									stSlideNest.State				:= E_SlideNest_State.READY;									
									bNestLeft						:= FALSE;
																	
								END_IF
	
	
	E_SlideNest_State.READY:
	
								IF stSlideNest.CMD.bExecute AND 	stSlideNest.CMD.SlideCylinderCMD.MoveRight	THEN

									stSlideNest.State				:= E_SlideNest_State.MOVE_RIGHT;
									
								ELSIF stSlideNest.CMD.bExecute AND 	stSlideNest.CMD.SlideCylinderCMD.MoveLeft	THEN
									
									stSlideNest.State				:= E_SlideNest_State.MOVE_LEFT;									
																		
								END_IF
	

	E_SlideNest_State.MOVE_RIGHT:
	
								bNestRight							:= TRUE;
								
								IF bNestInRightPos	THEN
									
									stSlideNest.State				:= E_SlideNest_State.DONE;
								
								END_IF
								
	E_SlideNest_State.MOVE_LEFT:
	
								bNestLeft							:= TRUE;
								
								IF bNestInLeftPos THEN
									
									stSlideNest.State				:= E_SlideNest_State.DONE;
								
								END_IF
								
	E_SlideNest_State.DONE:
	
	
								IF stSlideNest.CMD.bAcknowledge THEN
									
									stSlideNest.CMD.bAcknowledge	:= FALSE;
									stSlideNest.State				:= E_SlideNest_State.RESET;
								
								END_IF
	
	
	E_SlideNest_State.RESET:	
	
								bNestRight							:= FALSE;
								bNestLeft							:= FALSE;
								
								IF NOT stSlideNest.CMD.bAbort AND NOT stSlideNest.CMD.bEndCycle THEN
									
									stSlideNest.State				:= E_SlideNest_State.READY;
									
								ELSE stSlideNest.State			:= E_SlideNest_State.ABORTED;
								END_IF
									

ELSE stSlideNest.State		:= E_SlideNest_State.ABORTED;
	
END_CASE
/////////////////////////////////////////////////////////////////////////////////////STATUS/////////////////////////////////////////////////////////////////////////////////////

stSlideNest.Status.bBusy			:= 	stSlideNest.State	= E_SlideNest_State.MOVE_RIGHT OR
										stSlideNest.State	= E_SlideNest_State.MOVE_LEFT OR 
										stSlideNest.State	= E_SlideNest_State.STOPPING;
								
stSlideNest.Status.bDone			:=	stSlideNest.State	= E_SlideNest_State.DONE;

stSlideNest.Status.bReady			:= 	stSlideNest.State	= E_SlideNest_State.READY;

stSlideNest.Status.bStopped		:= 	NOT stSlideNest.Status.bBusy;
END_ACTION

ACTION b_ACT_IO_B:

bNestInLeftPos									:= dw_T08_EL1809.iSlideNestRetracted;
bNestInRightPos									:= dw_T08_EL1809.iSlideNestExtended; 

dw_T09_EL2809.qExtendSlideNest					:= bNestRight OR bSlideNestRight;	
dw_T09_EL2809.qRetractSlideNest					:= bNestLeft OR bSlideNestLeft;

bProcessCylinderUp								:= stTwinSAFE.qProcessCylinderRetracted;
END_ACTION

ACTION d_ACT_Set_Events_Station_4B:
//IMMEDIATE FAULTS

stStationEvents[4].aEvents[0].bEventTimer( IN :=  (bNestRight OR bSlideNestLeft) AND NOT bNestInLeftPos, PT := T#5S);
stStationEvents[4].aEvents[0].bFault						:= TRUE;
stStationEvents[4].aEvents[0].bEventFlag					:= stStationEvents[4].aEvents[0].bEventTimer.Q;
stStationEvents[4].aEvents[0].bEventText					:= 'Process Door extend timeout';
stStationEvents[4].aEvents[0].sSolution						:= 'Check cylinder, neumatic connections and sensors';

stStationEvents[4].aEvents[1].bEventTimer( IN :=  (bNestLeft OR bSlideNestRight) AND NOT bNestInRightPos, PT := T#5S);
stStationEvents[4].aEvents[1].bFault						:= TRUE;
stStationEvents[4].aEvents[1].bEventFlag					:= stStationEvents[4].aEvents[1].bEventTimer.Q;
stStationEvents[4].aEvents[1].bEventText					:= 'Process Door Retract timeout';
stStationEvents[4].aEvents[1].sSolution						:= 'Check cylinder, neumatic connections and sensors';
END_ACTION

END_PROGRAM

// ---- POUs/A_MASTER/A_2_PRG_MachineCtrl.TcPOU
PROGRAM A_2_PRG_MachineCtrl
VAR
/////////////////////////////////////////////////////////////////////////////////////TIMERS & TRIGGERS/////////////////////////////////////////////////////////////////////////////////////

	tonSys_Init					: Tc2_Standard.TON:=(PT:=T#1S);
	tonSys_InitTimeout			: Tc2_Standard.TON:=(PT:=T#15S);					
	tonFirstAutoCycle			: Tc2_Standard.TON:=(PT:=T#500MS);
	tonStopped					: TON := (PT := T#500MS);
	
/////////////////////////////////////////////////////////////////////////////////////PROCESS CYCLE/////////////////////////////////////////////////////////////////////////////////////	
	
	eCycleState					: E_General_ProcessCycle;
	tonCMD_Done					: TON;
	tonResetAllCMD				: TON;
	tonExecute					: TON;
	tonSave_Data				: TON;
	tonWriteToCsv				: TON;
	rFirstAutoCycle				: R_TRIG;
	
	bStartProcessCondition		: BOOL;
	bLeakTestDoneFlag			: BOOL;
	bHeightTestDoneFlag			: BOOL;
	i							: INT;

	tonGettingResults			: TON;
	ctuRejectPart				: CTU;
	
	tonProcessCylinderDelay		: TON;
	tonSealing					: TON;
	
	tonCylinderDwell			: TON; //Renan added - Buglist n13 - 08Jul26
	
	

/////////////////////////////////////////////////////////////////////////////////////I/O/////////////////////////////////////////////////////////////////////////////////////	

	bSlideNestNotHomed			: BOOL;
	bPartPresentNest1			: BOOL;
	bPartPresentNest2			: BOOL;
	rRejectSensor				: R_TRIG;
	bTwoHandsSignal				: BOOL;
	tonTwoHandsSignal			: TON;
	
	bProcessedPart				: ARRAY[0..1] OF BOOL;
	fProcessedPart				: ARRAY[0..1] OF F_TRIG;
	
		(* Renan Added - Buglist n6 - 08Jul26 *)
	bNest1StartOK				: BOOL;
	bNest2StartOK				: BOOL;
	bCycleHasFailure 			: BOOL;
	bCycleAllProcessedPass		: BOOL;
	(*\Renan Added - Buglist n6 - 08Jul26 *)
	
	bPuckLockerReadyToStart		: BOOL; (* Renan Added - Puck Locker Bug - 08Jul26 *)
	nPucksToRelease 			: USINT;(* Renan Added - Puck Locker Bug - 08Jul26 *)
	bPuckLockerEnable       	: BOOL; (* Renan added - Puck Locker Bug - 10Jul26*)
	bTest						: BOOL;
	
	bBottomSealer				: BOOL;
	bTopSealer					: BOOL;
	
	
END_VAR

/////////////////////////////////////////////////////////////////////////////////////GENERAL/////////////////////////////////////////////////////////////////////////////////////
a_ACT_MachineStatus();
b_ACT_ProcessCycle();
d_ACT_IO();

ACTION a_ACT_MachineStatus:
/////////////////////////////////////////////////////////////////////////////////////Utilities/////////////////////////////////////////////////////////////////////////////////////
tonSys_Init(IN:=stMachineStatus.bInitialising);
tonSys_InitTimeout(IN:=stMachineStatus.bInitialising);
tonSafety( IN := stMachineStatus.eMachineState = E_MachineState.SAFETY, PT := T#10S);
tonStopped(IN := stMachineStatus.eMachineState = E_MachineState.STOPPED);
	
	IF stMachineStatus.eMachineState <> E_MachineState.SYSTEM_AUTO_CYCLE AND 
		stMachineStatus.eMachineState <> E_MachineState.SYSTEM_INITIALISING THEN
		
		sMachineMessage									:= '';			
		
	END_IF
	
	IF (stMachineStatus.eMachineState = E_MachineState.STOPPED)  OR 
		(stMachineStatus.eMachineState = E_MachineState.STOPPING) THEN
		
		stTwinSAFE.iMachineStopped						:= TRUE;
		stTwinSAFE.iRunSafety							:= FALSE;
	
	ELSIF (stMachineStatus.eMachineState = E_MachineState.SAFETY) OR (stMachineStatus.eMachineState = E_MachineState.SYSTEM_INITIALISING) OR 
		(stMachineStatus.eMachineState = E_MachineState.SYSTEM_READY_TO_START) OR (stMachineStatus.eMachineState = E_MachineState.SYSTEM_AUTO_CYCLE) 
		OR (stMachineStatus.eMachineState = E_MachineState.MANUAL_MODE)THEN

		stTwinSAFE.iRunSafety							:= TRUE;
		stTwinSAFE.iMachineStopped						:= FALSE;
	
	ELSE stTwinSAFE.iMachineStopped						:= FALSE;
		stTwinSAFE.iRunSafety							:= FALSE;
		
	END_IF
	
	IF stMachineStatus.eMachineState = E_MachineState.SAFETY THEN
		
		stTwinSAFE.iInitSafety							:= TRUE;
		
	ELSE stTwinSAFE.iInitSafety							:= FALSE;
		
	END_IF

/////////////////////////////////////////////////////////////////////////////////////CONDITIONS/////////////////////////////////////////////////////////////////////////////////////
				IF NOT stMasterCtrl.bNoFault THEN
					stMachineStatus.eMachineState 		:= E_MachineState.FAULT;
				END_IF
				
				IF stMachineStatus.eMachineState		= E_MachineState.STOPPING OR
				stMachineStatus.eMachineState			= E_MachineState.FAULT THEN
					
					stSlideNest.CMD.bAbort				:= TRUE;	
					stLeakTesters.CMD.bAbort			:= TRUE;	
					stHeightTests.CMD.bAbort			:= TRUE;
					stProcessCylinder.CMD.bAbort		:= TRUE;
					stProcessDoor.CMD.bAbort			:= TRUE;
				
					stSlideNest.CMD.bEnable				:= FALSE;	
					stLeakTesters.CMD.bEnable			:= FALSE;	
					stHeightTests.CMD.bEnable			:= FALSE;
					stProcessCylinder.CMD.bEnable		:= FALSE;
					stProcessDoor.CMD.bEnable			:= FALSE;
					
				END_IF
				
				IF 	stButtonsLamps.bResetButtonFallingEdge THEN
					stSlideNest.CMD.bReset				:= TRUE;	
					stLeakTesters.CMD.bReset			:= TRUE;	
					stHeightTests.CMD.bReset			:= TRUE;
					stProcessCylinder.CMD.bReset		:= TRUE;
					stProcessDoor.CMD.bReset			:= TRUE;
				ELSE 
					stSlideNest.CMD.bReset				:= FALSE;	
					stLeakTesters.CMD.bReset			:= FALSE;	
					stHeightTests.CMD.bReset			:= FALSE;
					stProcessCylinder.CMD.bReset		:= FALSE;
					stProcessDoor.CMD.bReset			:= FALSE;
				END_IF	

				IF 	NOT (stMachineStatus.eMachineState = E_MachineState.MANUAL_MODE) THEN
					
					stSlideNest.CMD.bManualMode				:=FALSE;
					stLeakTesters.CMD.bManualMode			:=FALSE;
					stHeightTests.CMD.bManualMode			:=FALSE;
					stProcessCylinder.CMD.bManualMode		:=FALSE;
					stProcessDoor.CMD.bManualMode			:=FALSE;
					
				END_IF
				
				IF stMachineStatus.eMachineState = E_MachineState.SYSTEM_POWER_UP THEN
					
					bReadAMSNetID							:= TRUE;
				
				ELSE 
					
					bReadAMSNetID							:= FALSE;
					
				END_IF
				
				IF stMachineStatus.eMachineState		= E_MachineState.FAULT THEN
					
					bOpenDoorCycleFault						:= TRUE;
					
				ELSE bOpenDoorCycleFault					:= FALSE;
					
				END_IF
				
/////////////////////////////////////////////////////////////////////////////////////MACHINE CONTROL/////////////////////////////////////////////////////////////////////////////////////

CASE stMachineStatus.eMachineState OF

E_MachineState.SYSTEM_POWER_UP: 		

				fbGetLocalAMSNetID.bExecute				:= TRUE;
				bLightsOnOff							:= TRUE;
				IF tonSystemPowerUP.Q THEN
						stMachineStatus.eMachineState 	:= E_MachineState.STOPPED;//
				END_IF
	
E_MachineState.STOPPED:		

				stTwinSAFE.iRunSafety					:= FALSE;				

				IF stMasterCtrl.bNoFault   AND NOT stMasterCtrl.bCycleStopRequest AND ftrigButton[3].Q AND tonStopped.Q THEN
						stMachineStatus.eMachineState 	:= E_MachineState.SAFETY;//
				ELSIF NOT stMasterCtrl.bNoFault    THEN	
					stMachineStatus.eMachineState 		:= E_MachineState.FAULT;		
				END_IF	

E_MachineState.SAFETY:

				GVL_IO.dw_T09_EL2809.qOpenProcessDoor   := TRUE; // Thays added - Buglist n1 - 08Jul26
				stTwinSAFE.iRunSafety					:= TRUE;
				
				IF stTwinSAFE.qSafetyOk THEN
					
					stMachineStatus.eMachineState		:= E_MachineState.SYSTEM_INITIALISING;
					
				ELSIF stButtonsLamps.bStopButtonFallingEdge OR  
				stMasterCtrl.bCycleStopRequest OR tonSys_InitTimeout.Q  THEN
				
					stMachineStatus.eMachineState 		:= E_MachineState.STOPPING;	
					
				ELSIF NOT stMasterCtrl.bNoFault THEN		
					
					stMachineStatus.eMachineState 		:= E_MachineState.FAULT;
	
				END_IF
								

E_MachineState.SYSTEM_INITIALISING:		
					
					
				stSlideNest.CMD.bAbort					:= FALSE;	
				stLeakTesters.CMD.bAbort				:= FALSE;	
				stHeightTests.CMD.bAbort				:= FALSE;
				stProcessCylinder.CMD.bAbort			:= FALSE;
				stProcessDoor.CMD.bAbort				:= FALSE;	

				IF ( NOT stTwinSAFE.qProcessCylinderRetracted OR bSlideNestNotHomed) AND NOT bProcessDoorClosed THEN
						
						sMachineMessage					:= 'trigger both safety buttons to reset machine';
						
						IF bTwoHandsSignal  THEN
							
							tonSys_InitTimeout.IN		:= TRUE;	
							stLeakTesters.CMD.bEnable	:= TRUE;	
							stHeightTests.CMD.bEnable	:= TRUE;
							stProcessCylinder.CMD.bEnable:= TRUE;
							stProcessDoor.CMD.bEnable	:= TRUE;
							stSlideNest.CMD.bEnable		:= TRUE;
							sMachineMessage				:= '';
							
						END_IF
				ELSIF stTwinSAFE.qProcessCylinderRetracted AND dw_T08_EL1809.iSlideNestRetracted THEN
					
					stSlideNest.CMD.bEnable				:= TRUE;	
					stLeakTesters.CMD.bEnable			:= TRUE;	
					stHeightTests.CMD.bEnable			:= TRUE;
					stProcessCylinder.CMD.bEnable		:= TRUE;
					stProcessDoor.CMD.bEnable			:= TRUE;				
				
				END_IF
				
				IF stMasterCtrl.bAllStationsReady  THEN 
					stMachineStatus.eMachineState		:= E_MachineState.SYSTEM_READY_TO_START;
				ELSIF stButtonsLamps.bStopButtonFallingEdge OR  
				stMasterCtrl.bCycleStopRequest OR tonSys_InitTimeout.Q  THEN
					stMachineStatus.eMachineState 		:= E_MachineState.STOPPING;	
				ELSIF NOT stMasterCtrl.bNoFault THEN		
					stMachineStatus.eMachineState 		:= E_MachineState.FAULT;
				END_IF
			
					
E_MachineState.SYSTEM_READY_TO_START:	

				IF 	 stButtonsLamps.bStartButtonFallingEdge AND stMasterCtrl.bAllStationsReady  THEN
					stMachineStatus.eMachineState 		:= E_MachineState.SYSTEM_AUTO_CYCLE;
				ELSIF NOT stMasterCtrl.bAllStationsReady OR stMasterCtrl.bCycleStopRequest THEN
					stMachineStatus.eMachineState 		:= E_MachineState.STOPPING;		
				ELSIF NOT stMasterCtrl.bNoFault THEN	
					stMachineStatus.eMachineState 		:= E_MachineState.FAULT;
				ELSIF GVL_Master.stMasterCTRL.bManualModeRequest AND stMasterCtrl.bNoFault THEN
					stMachineStatus.eMachineState 		:= E_MachineState.MANUAL_MODE;
				END_IF

				

E_MachineState.SYSTEM_AUTO_CYCLE:		

				
				IF  stMasterCtrl.bCycleStopRequest AND (eCycleState = E_General_ProcessCycle.IDLE) THEN
	
					stMachineStatus.eMachineState 		:= E_MachineState.STOPPING;
				
				ELSIF stMasterCtrl.bCycleStopRequest AND NOT (eCycleState = E_General_ProcessCycle.IDLE) THEN					
				
					sMachineMessage						:= 'Ending  Cycle';
				
				ELSIF NOT stMasterCtrl.bNoFault THEN	
					stMachineStatus.eMachineState 		:= E_MachineState.FAULT;
				END_IF
				

E_MachineState.STOPPING:	

				
				IF stMasterCtrl.bAllStationsStopped THEN
					stMachineStatus.eMachineState 		:= E_MachineState.STOPPED;
				ELSIF NOT stMasterCtrl.bNoFault THEN	
					stMachineStatus.eMachineState 		:= E_MachineState.FAULT;					
				END_IF
				
				stTwinSAFE.iRunSafety					:= FALSE;	

E_MachineState.FAULT:	
				
				GVL_IO.dw_T09_EL2809.qOpenProcessDoor   :=TRUE; // Thays added - Buglist n1 - 08Jul26

				IF stMasterCtrl.bNoFault	THEN
					stMachineStatus.eMachineState		:= E_MachineState.STOPPED;		
				END_IF
				
				stTwinSAFE.iRunSafety					:= FALSE;	

E_MachineState.MANUAL_MODE:

				IF stButtonsLamps.bStopButtonFallingEdge OR NOT GVL_Master.stMasterCTRL.bManualModeRequest THEN
					stMachineStatus.eMachineState 		:= E_MachineState.STOPPING;
				ELSIF  NOT stMasterCtrl.bNoFault THEN	
					stMachineStatus.eMachineState 		:= E_MachineState.FAULT;								
				ELSE 
					
					stSlideNest.CMD.bManualMode				:=TRUE;
					stLeakTesters.CMD.bManualMode			:=TRUE;
					stHeightTests.CMD.bManualMode			:=TRUE;
					stProcessCylinder.CMD.bManualMode		:=TRUE;
					stProcessDoor.CMD.bManualMode			:=TRUE;

				END_IF
				
					
ELSE
stMachineStatus.eMachineState:=E_MachineState.SYSTEM_POWER_UP;		
END_CASE									


/////////////////////////////////////////////////////////////////////////////////////MACHINE STATUS/////////////////////////////////////////////////////////////////////////////////////
stMachineStatus.bSystemPowerUp 			:= (stMachineStatus.eMachineState = E_MachineState.SYSTEM_POWER_UP);
stMachineStatus.bStopped 				:= (stMachineStatus.eMachineState = E_MachineState.STOPPED);
stMachineStatus.bInitialising 			:= (stMachineStatus.eMachineState = E_MachineState.SYSTEM_INITIALISING);
stMachineStatus.bReadyToStart 			:= (stMachineStatus.eMachineState = E_MachineState.SYSTEM_READY_TO_START);
stMachineStatus.bAutoCycle 				:= (stMachineStatus.eMachineState = E_MachineState.SYSTEM_AUTO_CYCLE);
stMachineStatus.bStopping 				:= (stMachineStatus.eMachineState = E_MachineState.STOPPING);
stMachineStatus.bFault 					:= (stMachineStatus.eMachineState = E_MachineState.FAULT);
stMachineStatus.bManualMode 			:= (stMachineStatus.eMachineState = E_MachineState.MANUAL_MODE);
stMachineStatus.bSafety 				:= (stMachineStatus.eMachineState = E_MachineState.SAFETY);

/////////////////////////////////////////////////////////////////////////////////////FLAGS/////////////////////////////////////////////////////////////////////////////////////
stMasterCtrl.bAllStationsStopped		:= stSlideNest.Status.bStopped AND stLeakTesters.Status.bStopped AND stHeightTests.Status.bStopped AND stProcessCylinder.Status.bStopped AND stProcessDoor.Status.bStopped AND
										   NOT stSlideNest.Status.bBusy AND NOT stLeakTesters.Status.bBusy AND NOT stHeightTests.Status.bBusy AND NOT stProcessCylinder.Status.bBusy AND NOT stProcessDoor.Status.bBusy;
										   
stMasterCtrl.bAllStationsReady			:= stSlideNest.Status.bReady  AND stLeakTesters.Status.bReady AND stHeightTests.Status.bReady AND stProcessCylinder.Status.bReady AND stProcessDoor.Status.bReady;
END_ACTION

ACTION b_ACT_ProcessCycle:
/////////////////////////////////////////////////////////////////////////////////////UTILITIES & TRIGGERS/////////////////////////////////////////////////////////////////////////////////////
//ADD REJECT SENSOR FUNCTION. IF PART FAIL WE SHOULD WAIT UNTIL THE OPERATOR LEAVE THE FAIL PART IN THE CONTAINER

tonProcessCylinderDelay(IN := eCycleState = E_General_ProcessCycle.WAIT_CLOSE_PROCESS_DOOR, PT := T#100MS);

ctuRejectPart();
IF eCycleState = E_General_ProcessCycle.RESET_ALL_CMD THEN
	
	ctuRejectPart.RESET															:= TRUE;

ELSE ctuRejectPart.RESET														:= FALSE;	
	
END_IF
IF eCycleState = E_General_ProcessCycle.IDLE THEN
	
	bAutocycleIDLE																:= TRUE;
	
ELSE bAutocycleIDLE																:= FALSE;

END_IF
tonSealing(PT := T#1000MS);
tonGettingResults( IN := eCycleState = E_General_ProcessCycle.WAIT_RESULTS, PT := T#100MS);

tonCMD_Done( IN := , PT := T#500MS);
tonSave_Data( IN :=  eCycleState = E_General_ProcessCycle.SAVE_DATA2, PT := T#500MS);
tonResetAllCMD( IN := eCycleState = E_General_ProcessCycle.RESET_ALL_CMD, PT := T#500MS);


tonExecute( IN := 	eCycleState = E_General_ProcessCycle.CLOSE_PROCESS_DOOR OR
					eCycleState = E_General_ProcessCycle.OPEN_PROCESS_DOOR OR
					eCycleState = E_General_ProcessCycle.EXTEND_PROCESS_CYLINDER OR
					eCycleState = E_General_ProcessCycle.RETRACT_PROCESS_CYLINDER OR
					eCycleState = E_General_ProcessCycle.RETRACT_MIDDLE_PROCESS_CYLINDER OR
					eCycleState = E_General_ProcessCycle.WAIT_PRE_RETRACT_PROCESS_CYLINDER OR
					eCycleState = E_General_ProcessCycle.MOVE_NEST_TO_RIGHT OR
					eCycleState = E_General_ProcessCycle.MOVE_NEST_TO_LEFT OR
					eCycleState = E_General_ProcessCycle.LEAK_TEST OR
					eCycleState = E_General_ProcessCycle.HEIGHT_TEST OR
					eCycleState = E_General_ProcessCycle.WAIT_TO_SAVE_DATA,
					PT := T#500MS);
					
tonCylinderDwell( IN := eCycleState = E_General_ProcessCycle.PRE_RETRACT_PROCESS_CYLINDER, PT := T#250MS);
					
IF (stMachineStatus.eMachineState <> E_MachineState.SYSTEM_AUTO_CYCLE) THEN
	
	eCycleState																	:= E_General_ProcessCycle.RESET_ALL_CMD;

END_IF

rFirstAutoCycle( CLK := stMachineStatus.bAutoCycle);

IF (eCycleState = E_General_ProcessCycle.LEAK_TEST) OR (eCycleState = E_General_ProcessCycle.HEIGHT_TEST) THEN
	
			sMachineMessage														:= 'Inspection in process ';

END_IF

IF stMachineStatus.eMachineState <> E_MachineState.SYSTEM_AUTO_CYCLE THEN
	
	MEMSET( destAddr := ADR(stCycleDataNest1), fillByte := 0, n := SIZEOF(stCycleDataNest1));
	MEMSET( destAddr := ADR(stCycleDataNest2), fillByte := 0, n := SIZEOF(stCycleDataNest2));

END_IF

(* Renan Added 10Jul26*)
bPuckLockerEnable := GVL_HMI.bPuckLockerGateEnable;
(*\Renan Added 10Jul26*)

(*Renan added - Puck Locker Bug - 08Jul26*)
bPuckLockerReadyToStart := (NOT bPuckLockerEnable) OR (GVL_Stations.stPuckLocker.bPuckDetected AND
							GVL_Stations.stPuckLocker.bPuckLocked AND GVL_Stations.stPuckLocker.eState = E_PuckLockerState.Locked);
(*\Renan added - Puck Locker Bug - 08Jul26*)

(*Renan Added 06Jul26*)
IF bPuckLockerEnable THEN
	GVL_Stations.stPuckLocker.bNestsEmpty := ((NOT bProcessedPart[0]) OR (NOT bPartPresentNest1)) AND ((NOT bProcessedPart[1]) OR (NOT bPartPresentNest2));
ELSE
	GVL_Stations.stPuckLocker.bNestsEmpty := TRUE;
END_IF
(*\Renan Added 06Jul26*)

	
/////////////////////////////////////////////////////////////////////////////////////CONDITIONS/////////////////////////////////////////////////////////////////////////////////////

(* Renan Added - Buglist n6 - 08Jul26 *)
bNest1StartOK := (NOT bNest1Flag) OR bPartPresentNest1;
bNest2StartOK := (NOT bNest2Flag) OR bPartPresentNest2;
(*\Renan Added - Buglist n6 - 08Jul26 *)

bStartProcessCondition := bTwoHandsSignal AND (bPartPresentNest1 OR NOT bNest1Flag) AND (bPartPresentNest2 OR NOT bNest2Flag) AND (bNest1Flag OR bNest2Flag);



IF rFirstAutoCycle.Q THEN
	eCycleState																	:= E_General_ProcessCycle.RESET_ALL_CMD;
END_IF


CASE eCycleState OF
	
E_General_ProcessCycle.RESET_ALL_CMD:

				stProcessDoor.CMD.ProcessDoorCMD.OpenDoor						:= FALSE;
				stProcessDoor.CMD.ProcessDoorCMD.CloseDoor						:= FALSE;
				stProcessDoor.CMD.bExecute										:= FALSE;
				
				stProcessCylinder.CMD.ProcessCylinderCMD.ExtendCylinder			:= FALSE;
				stProcessCylinder.CMD.ProcessCylinderCMD.RetractCylinder		:= FALSE;
				stProcessCylinder.CMD.bExecute									:= FALSE;
				
				stLeakTesters.CMD.LeakTestersCMD.RunLeakTester1					:= FALSE;
				stLeakTesters.CMD.LeakTestersCMD.RunLeakTester2					:= FALSE;
				stLeakTesters.CMD.bExecute										:= FALSE;
				
				stHeightTests.CMD.HeightTest_CMD.Measurement1					:= FALSE;
				stHeightTests.CMD.HeightTest_CMD.Measurement2					:= FALSE;
				stHeightTests.CMD.bExecute										:= FALSE;
				
				stSlideNest.CMD.SlideCylinderCMD.MoveLeft						:= FALSE;
				stSlideNest.CMD.SlideCylinderCMD.MoveRight						:= FALSE;
				
				bWriteNest1														:= FALSE;
				bWriteNest2														:= FALSE;
				bRejectPartDialog[0]											:= FALSE;
				bRejectPartDialog[1]											:= FALSE;
				bRejectPartFault												:= FALSE;
				
				bHeightTestDoneFlag												:= FALSE;
				bLeakTestDoneFlag												:= FALSE;
				
				bProcessedPart[0]												:= FALSE;
				bProcessedPart[1]												:= FALSE;
				
				bTopSealer														:= FALSE;
				bBottomSealer													:= FALSE;
				tonSealing.IN													:= FALSE;
			
				//add reset command to reset all cycle data
				
				IF tonResetAllCMD.Q AND stMachineStatus.bAutoCycle THEN
					
					eCycleState													:= E_General_ProcessCycle.IDLE;		
				
				END_IF
	
E_General_ProcessCycle.IDLE:
		
				//start cycle
				IF bStartProcessCondition AND NOT bProcessedPart[0] AND NOT bProcessedPart[1] AND bPuckLockerReadyToStart THEN (*Renan added - Puck Locker Bug - 08Jul26*) //Original: IF bStartProcessCondition AND NOT bProcessedPart[0] AND NOT bProcessedPart[1] THEN
					
					MEMSET( destAddr := ADR(stCycleDataNest1), fillByte := 0, n := SIZEOF(stCycleDataNest1));
					MEMSET( destAddr := ADR(stCycleDataNest2), fillByte := 0, n := SIZEOF(stCycleDataNest2));
					
					IF bNest1Flag THEN
						
						bProcessedPart[0]										:= bPartPresentNest1;
						
					END_IF
					
					IF bNest2Flag THEN
						
						bProcessedPart[1]										:= bPartPresentNest2;
						
					END_IF
					
					eCycleState													:= E_General_ProcessCycle.CLOSE_PROCESS_DOOR;
					
				END_IF
				
				IF bPuckLockerEnable AND NOT bPuckLockerReadyToStart AND NOT bProcessedPart[0] AND NOT bProcessedPart[1] THEN
				
					IF NOT GVL_Stations.stPuckLocker.bPuckDetected THEN
						
						sMachineMessage 		:= 'Insert puck into locker to continue';
						
					ELSE
						
						sMachineMessage := 'Waiting for puck locker to lock puck';
						
					END_IF					
				
				ELSIF  bPuckLockerReadyToStart AND (bPartPresent[0] OR NOT bNest1Flag) AND (bPartPresent[1] OR NOT bNest2Flag) THEN
					
					sMachineMessage := 'trigger both safety buttons to start cycle';
					
				ELSIF bPuckLockerReadyToStart AND ( (NOT bPartPresent[0] AND bNest1Flag) AND (NOT bPartPresent[1] AND bNest2Flag)) THEN
					
					sMachineMessage 			:= 'Place parts to continue';
					
				ELSIF bPuckLockerReadyToStart AND ( (bPartPresent[0] OR NOT bNest1Flag) AND (NOT bPartPresent[1] AND bNest2Flag)) THEN
					
					sMachineMessage 			:= 'Place part in nest 2 to continue';
				
				ELSIF bPuckLockerReadyToStart AND ( (NOT bPartPresent[0] AND bNest1Flag) AND (bPartPresent[1] OR NOT bNest2Flag)) THEN
					
					sMachineMessage 			:= 'Place part in nest 1 to continue';
					
				END_IF
				
				
				//Messages to start cycle
				
					
				(* Renan added - Puck Locker Messages - 08Jul26 *)
				(*
				IF bPuckLockerEnable
				AND GVL_Stations.stPuckLocker.eState = E_PuckLockerState.WaitingForNestsEmpty THEN
				
					IF bPartPresentNest1 OR bPartPresentNest2 THEN
						
						sMachineMessage := 'Remove parts from nests to release puck';
						
					ELSE
						
						sMachineMessage := 'Waiting for puck to be released';
						
					END_IF
				
				ELSIF bProcessedPart[0] AND NOT bProcessedPart[1] AND NOT bStartProcessCondition THEN
					
					IF bPuckLockerEnable THEN
						sMachineMessage := 'Remove processed part from nest 1 to release puck';
					ELSE
						sMachineMessage := 'Remove Processed part from nest 1';
					END_IF
					
				ELSIF NOT bProcessedPart[0] AND bProcessedPart[1] AND NOT bStartProcessCondition THEN 
					
					IF bPuckLockerEnable THEN
						sMachineMessage := 'Remove processed part from nest 2 to release puck';
					ELSE
						sMachineMessage := 'Remove Processed part from nest 2';
					END_IF
					
				ELSIF bProcessedPart[0] AND bProcessedPart[1] AND NOT bStartProcessCondition THEN 
					
					IF bPuckLockerEnable THEN
						sMachineMessage := 'Remove processed parts to release puck';
					ELSE
						sMachineMessage := 'Remove Processed parts';
					END_IF
				
				ELSIF bPuckLockerEnable AND NOT bPuckLockerReadyToStart AND NOT bProcessedPart[0] AND NOT bProcessedPart[1] THEN
				
					IF NOT GVL_Stations.stPuckLocker.bPuckDetected THEN
						
						sMachineMessage := 'Insert puck into locker to continue';
						
					ELSE
						
						sMachineMessage := 'Waiting for puck locker to lock puck';
						
					END_IF
				
				ELSIF NOT bProcessedPart[0] AND NOT bProcessedPart[1] AND (NOT bPartPresentNest1 OR NOT bPartPresentNest2) THEN 
					
					sMachineMessage := 'Insert parts to continue';
				
				ELSIF NOT bProcessedPart[0] AND NOT bProcessedPart[1] AND bPartPresentNest1 AND bPartPresentNest2 THEN 
					
					sMachineMessage := 'trigger both safety buttons to start cycle';
				
				ELSE 
					
					sMachineMessage := '';
						
				END_IF*)
				(*\Renan added - Puck Locker Messages - 08Jul26*)
			
E_General_ProcessCycle.CLOSE_PROCESS_DOOR:

				stProcessDoor.CMD.ProcessDoorCMD.CloseDoor						:= TRUE;
				stProcessDoor.CMD.bExecute										:= TRUE;
				
				IF tonExecute.Q THEN
					
					eCycleState													:= E_General_ProcessCycle.WAIT_CLOSE_PROCESS_DOOR;	
					
				END_IF

E_General_ProcessCycle.WAIT_CLOSE_PROCESS_DOOR:
				
				IF stProcessDoor.Status.bDone AND tonProcessCylinderDelay.Q THEN
					
				stProcessDoor.CMD.ProcessDoorCMD.CloseDoor						:= FALSE;
				stProcessDoor.CMD.bExecute										:= FALSE;
				stProcessDoor.CMD.bAcknowledge									:= TRUE;
				eCycleState														:= E_General_ProcessCycle.PRE_RETRACT_PROCESS_CYLINDER;
				
				END_IF
		
E_General_ProcessCycle.PRE_RETRACT_PROCESS_CYLINDER:		

				stProcessCylinder.CMD.ProcessCylinderCMD.RetractCylinder		:= TRUE;	
				stProcessCylinder.CMD.bExecute			:= TRUE;
				
				IF tonCylinderDwell.Q THEN
					eCycleState							:= E_General_ProcessCycle.WAIT_PRE_RETRACT_PROCESS_CYLINDER;	
				END_IF

E_General_ProcessCycle.WAIT_PRE_RETRACT_PROCESS_CYLINDER:

				IF 	stProcessCylinder.Status.bDone OR stProcessCylinder.Status.bReady THEN
					
					stProcessCylinder.CMD.ProcessCylinderCMD.RetractCylinder		:= FALSE;
					stProcessCylinder.CMD.bExecute		:= FALSE;
					stProcessCylinder.CMD.bAcknowledge	:= TRUE;
					
					IF tonExecute.Q THEN
						eCycleState							:= E_General_ProcessCycle.EXTEND_PROCESS_CYLINDER;
					END_IF	
				END_IF
								
E_General_ProcessCycle.EXTEND_PROCESS_CYLINDER:
				
						
				stProcessCylinder.CMD.ProcessCylinderCMD.ExtendCylinder			:= TRUE;
				stProcessCylinder.CMD.bExecute									:= TRUE;
	
				IF tonExecute.Q THEN
					
					eCycleState													:= E_General_ProcessCycle.WAIT_EXTEND_PROCESS_CYLINDER;	
					
				END_IF

E_General_ProcessCycle.WAIT_EXTEND_PROCESS_CYLINDER:
			
				IF stProcessCylinder.Status.bDone THEN
					
					stProcessCylinder.CMD.ProcessCylinderCMD.ExtendCylinder		:= FALSE;
					stProcessCylinder.CMD.bExecute								:= FALSE;
					
					IF bHeightTestDoneFlag	THEN
						tonSealing.IN											:= TRUE;
						bTopSealer												:= TRUE;	
						IF tonSealing.Q THEN
							
							bBottomSealer										:= TRUE;
							tonSealing.IN										:= FALSE;
							stProcessCylinder.CMD.bAcknowledge					:= TRUE;
							eCycleState											:= E_General_ProcessCycle.WAIT_LEAK_TEST;
							
						END_IF	
					
					ELSE 

						eCycleState												:= E_General_ProcessCycle.HEIGHT_TEST;
						stProcessCylinder.CMD.bAcknowledge						:= TRUE;
						
					END_IF							
					
						
										
				END_IF
			   

E_General_ProcessCycle.HEIGHT_TEST:

				stHeightTests.CMD.HeightTest_CMD.Measurement1				 	:= bNest1Flag;
				stHeightTests.CMD.HeightTest_CMD.Measurement2				 	:= bNest2Flag;
				stHeightTests.CMD.bExecute										:= TRUE;
					
				IF tonExecute.Q THEN
					
					eCycleState													:= E_General_ProcessCycle.WAIT_HEIGHT_TEST;	
					
				END_IF

E_General_ProcessCycle.WAIT_HEIGHT_TEST:

				IF stHeightTests.Status.bDone THEN
					
					stHeightTests.CMD.HeightTest_CMD.Measurement1				:= FALSE;
					stHeightTests.CMD.HeightTest_CMD.Measurement2				:= FALSE;
					stHeightTests.CMD.bExecute									:= FALSE;
					stHeightTests.CMD.bAcknowledge 								:= TRUE;	
					bHeightTestDoneFlag											:= TRUE;
					eCycleState													:= E_General_ProcessCycle.LEAK_TEST;
					
				END_IF
(*			
E_General_ProcessCycle.RETRACT_MIDDLE_PROCESS_CYLINDER:
				
						
				stProcessCylinder.CMD.ProcessCylinderCMD.RetractCylinderMiddle	:= TRUE;
				stProcessCylinder.CMD.bExecute									:= TRUE;
	
				IF tonExecute.Q THEN
					
					eCycleState													:= E_General_ProcessCycle.WAIT_RETRACT_MIDDLE_PROCESS_CYLINDER;	
					
				END_IF

E_General_ProcessCycle.WAIT_RETRACT_MIDDLE_PROCESS_CYLINDER:
			
				IF stProcessCylinder.Status.bDone THEN
					
					stProcessCylinder.CMD.ProcessCylinderCMD.RetractCylinderMiddle	:= FALSE;
					stProcessCylinder.CMD.bExecute								:= FALSE;
					stProcessCylinder.CMD.bAcknowledge							:= TRUE;
												
					eCycleState													:= E_General_ProcessCycle.MOVE_NEST_TO_RIGHT;	
						
										
				END_IF
*)

E_General_ProcessCycle.LEAK_TEST:

				stLeakTesters.CMD.LeakTestersCMD.RunLeakTester1					:= bNest1Flag;
				stLeakTesters.CMD.LeakTestersCMD.RunLeakTester2					:= bNest2Flag;
				stLeakTesters.CMD.bExecute										:= TRUE;
				
				IF tonExecute.Q THEN
					
					eCycleState													:= E_General_ProcessCycle.RETRACT_PROCESS_CYLINDER;	
					
				END_IF
				
E_General_ProcessCycle.MOVE_NEST_TO_RIGHT:		

				stSlideNest.CMD.SlideCylinderCMD.MoveRight						:= TRUE;
				stSlideNest.CMD.bExecute										:= TRUE;
	
				IF tonExecute.Q THEN
					
					eCycleState													:= E_General_ProcessCycle.WAIT_MOVE_NEST_TO_RIGHT;	
					
				END_IF	
				
E_General_ProcessCycle.WAIT_MOVE_NEST_TO_RIGHT:
			
				IF stSlideNest.Status.bDone THEN
					
					stSlideNest.CMD.SlideCylinderCMD.MoveRight					:= FALSE;
					stSlideNest.CMD.bExecute									:= FALSE;
					stSlideNest.CMD.bAcknowledge								:= TRUE;
												
					eCycleState													:= E_General_ProcessCycle.EXTEND_PROCESS_CYLINDER;	
						
										
				END_IF
	

E_General_ProcessCycle.WAIT_LEAK_TEST:

				IF stLeakTesters.Status.bDone THEN
					
					stLeakTesters.CMD.bExecute									:= FALSE;
					stLeakTesters.CMD.LeakTestersCMD.RunLeakTester1				:= FALSE;
					stLeakTesters.CMD.LeakTestersCMD.RunLeakTester2				:= FALSE;
					stLeakTesters.CMD.bAcknowledge 								:= TRUE;	
					bLeakTestDoneFlag											:= TRUE;
					eCycleState													:= E_General_ProcessCycle.WAIT_RESULTS;
					
				END_IF
				
E_General_ProcessCycle.WAIT_RESULTS:

				IF tonGettingResults.Q THEN
					
					eCycleState													:= E_General_ProcessCycle.RESULTS;
					
				END_IF


E_General_ProcessCycle.RESULTS:

				
					
					IF bProcessedPart[0] THEN
					
						IF stCycleDataNest1.LeakTest_Pass AND stCycleDataNest1.HeightTest_Pass THEN	
				
							stCycleDataNest1.bPass								:= TRUE;
							stCycleDataNest1.bFail								:= FALSE;
				
						ELSE stCycleDataNest1.bFail								:= TRUE;
							stCycleDataNest1.bPass								:= FALSE;
				
						END_IF
					
					END_IF
				
					IF bProcessedPart[1] THEN
					
						IF stCycleDataNest2.LeakTest_Pass AND stCycleDataNest2.HeightTest_Pass THEN	
				
							stCycleDataNest2.bPass								:= TRUE;
							stCycleDataNest2.bFail								:= FALSE;
				
						ELSE stCycleDataNest2.bFail								:= TRUE;
							stCycleDataNest2.bPass								:= FALSE;
				
						END_IF
					
					END_IF
					
				
				
				
				
				stCycleDataNest1.sTime											:= sSystemTime;
				stCycleDataNest1.sDate											:= sSystemDate;
				stCycleDataNest2.sTime											:= sSystemTime;
				stCycleDataNest2.sDate											:= sSystemDate;
					
				eCycleState														:= E_General_ProcessCycle.WAIT_TO_SAVE_DATA;
									
E_General_ProcessCycle.WAIT_TO_SAVE_DATA:
				
				IF tonExecute.Q THEN
					
					eCycleState													:= E_General_ProcessCycle.SAVE_DATA;	
					
				END_IF

E_General_ProcessCycle.SAVE_DATA:

				IF bProcessedPart[0] THEN
					
					FOR i := 199 TO 0 BY -1 DO
						
						aDataHistoryNest1[i+1] 									:= aDataHistoryNest1[i];
						
					END_FOR
				
				END_IF
				
				IF bProcessedPart[1] THEN
					
					FOR i := 199 TO 0 BY -1 DO
						
						aDataHistoryNest2[i+1] 									:= aDataHistoryNest2[i];
						
					END_FOR
				
				END_IF		
			
				eCycleState														:= E_General_ProcessCycle.SAVE_DATA2;
					
E_General_ProcessCycle.SAVE_DATA2:	
				
				
				c_ACT_SaveData();	
								
				eCycleState														:= E_General_ProcessCycle.CSV_NEST1;
				
				
E_General_ProcessCycle.CSV_NEST1:

				IF bProcessedPart[0] THEN
					
					bWriteNest1													:= TRUE;
					
					IF bCSVDone OR bCSVError THEN
						
						eCycleState												:= E_General_ProcessCycle.CSV_NEST2;
						bWriteNest1												:= FALSE;
						bCSVError												:= FALSE;
						
					END_IF
					
				ELSE eCycleState												:= E_General_ProcessCycle.CSV_NEST2;				
					
				END_IF
			
				
E_General_ProcessCycle.CSV_NEST2:

				IF bCSVDone THEN
					
						bWriteNest2												:= FALSE;
						eCycleState												:= E_General_ProcessCycle.RETRACT_PROCESS_CYLINDER;	
	
				END_IF

				IF bProcessedPart[1] AND  bCSVReady AND NOT bCSVDone AND NOT bCSVError THEN
				
						bWriteNest2												:= TRUE;

				ELSIF NOT bProcessedPart[1] OR bCSVError THEN

						 eCycleState											:= E_General_ProcessCycle.RETRACT_PROCESS_CYLINDER;
						 bCSVError												:= FALSE;
						 
				END_IF
				
				
					
				
E_General_ProcessCycle.RETRACT_PROCESS_CYLINDER:
						
				stProcessCylinder.CMD.ProcessCylinderCMD.RetractCylinder		:= TRUE;	
				stProcessCylinder.CMD.bExecute									:= TRUE;
				bTopSealer														:= FALSE;
				bBottomSealer													:= FALSE;
				
				IF tonExecute.Q THEN
					
					eCycleState													:= E_General_ProcessCycle.WAIT_RETRACT_PROCESS_CYLINDER;	
					
				END_IF

E_General_ProcessCycle.WAIT_RETRACT_PROCESS_CYLINDER:

				IF 	stProcessCylinder.Status.bDone THEN
					
					stProcessCylinder.CMD.ProcessCylinderCMD.RetractCylinder	:= FALSE;
					stProcessCylinder.CMD.bExecute								:= FALSE;
					stProcessCylinder.CMD.bAcknowledge							:= TRUE;
					
					IF bLeakTestDoneFlag THEN
						
						eCycleState												:= E_General_ProcessCycle.MOVE_NEST_TO_LEFT;
						
					ELSE 	eCycleState											:= E_General_ProcessCycle.MOVE_NEST_TO_RIGHT;
					END_IF
					
					
					
				END_IF

E_General_ProcessCycle.MOVE_NEST_TO_LEFT:		

				stSlideNest.CMD.SlideCylinderCMD.MoveLeft						:= TRUE;
				stSlideNest.CMD.bExecute										:= TRUE;
	
				IF tonExecute.Q THEN
					
					eCycleState													:= E_General_ProcessCycle.WAIT_MOVE_NEST_TO_LEFT;	
					
				END_IF	
				
E_General_ProcessCycle.WAIT_MOVE_NEST_TO_LEFT:
			
				IF stSlideNest.Status.bDone THEN
					
					stSlideNest.CMD.SlideCylinderCMD.MoveLeft					:= FALSE;
					stSlideNest.CMD.bExecute									:= FALSE;
					stSlideNest.CMD.bAcknowledge								:= TRUE;
												
					IF NOT bEmptyRejectChute THEN

						eCycleState							:= E_General_ProcessCycle.OPEN_PROCESS_DOOR;
					
					ELSE eCycleState							:= E_General_ProcessCycle.REJECT_CHUTE_FULL; 
					
					END_IF
						
										
				END_IF
	
E_General_ProcessCycle.REJECT_CHUTE_FULL:

				sMachineMessage									:= 'Waiting for Reject chute empty';

				IF NOT bEmptyRejectChute THEN
					
						sMachineMessage							:= '';
						eCycleState								:= E_General_ProcessCycle.OPEN_PROCESS_DOOR;
				
				END_IF	
		
E_General_ProcessCycle.OPEN_PROCESS_DOOR:

				stProcessDoor.CMD.ProcessDoorCMD.OpenDoor						:= TRUE;
				stProcessDoor.CMD.bExecute										:= TRUE;
				
				IF tonExecute.Q THEN
					
					eCycleState													:= E_General_ProcessCycle.WAIT_OPEN_PROCESS_DOOR;	
					
				END_IF

E_General_ProcessCycle.WAIT_OPEN_PROCESS_DOOR:

				IF 	stProcessDoor.Status.bDone THEN
					
					stProcessDoor.CMD.ProcessDoorCMD.OpenDoor					:= FALSE;
					stProcessDoor.CMD.bExecute									:= FALSE;
					stProcessDoor.CMD.bAcknowledge								:= TRUE;
					
					eCycleState							:= E_General_ProcessCycle.PUCK_DEFINITION;
			
				
				END_IF
				
E_General_ProcessCycle.PUCK_DEFINITION:
		
				(* Renan Added - Buglist n6 - 08Jul26 *)
				bCycleHasFailure := (bProcessedPart[0] AND stCycleDataNest1.bFail) OR (bProcessedPart[1] AND stCycleDataNest2.bFail);

				bCycleAllProcessedPass := (bProcessedPart[0] OR bProcessedPart[1]) AND ((NOT bProcessedPart[0]) OR stCycleDataNest1.bPass) AND ((NOT bProcessedPart[1]) OR stCycleDataNest2.bPass);
					(*\Renan Added - Buglist n6 - 08Jul26 *)
					
					(* Renan Added 10Jul26 - Puck Locker *)
				IF bPuckLockerEnable AND bCycleAllProcessedPass THEN
					
					GVL_Stations.stPuckLocker.nRequestedRelease := USINT#0;
					
					IF bProcessedPart[0] AND stCycleDataNest1.bPass THEN
						
						GVL_Stations.stPuckLocker.nRequestedRelease := GVL_Stations.stPuckLocker.nRequestedRelease + USINT#1;
						
					END_IF
					
					IF bProcessedPart[1] AND stCycleDataNest2.bPass THEN
						
						GVL_Stations.stPuckLocker.nRequestedRelease := GVL_Stations.stPuckLocker.nRequestedRelease + USINT#1;
							
					END_IF
					
					GVL_Stations.stPuckLocker.bApplyDisposition := TRUE;
					
				END_IF
				
				
				IF bCycleHasFailure THEN //Bugfix 08Jul26
					
					eCycleState								:= E_General_ProcessCycle.WAIT_REJECT_PART;
					
				ELSIF bCycleAllProcessedPass THEN //Bugfix 08Jul26

					eCycleState								:= E_General_ProcessCycle.NEST_CLEARING;
						
				END_IF		
			
E_General_ProcessCycle.WAIT_REJECT_PART:
					
				ctuRejectPart.CU 								:= rRejectSensor.Q;				

				IF stCycleDataNest1.bFail AND NOT stCycleDataNest2.bFail THEN
					
					sMachineMessage												:= 'REMOVE PART FROM NEST 1 AND PUT IN REJECT CHUTE';
					
					IF ctuRejectPart.CV > 0 AND NOT bPartPresentNest1 AND (bPartPresentNest2 OR NOT bProcessedPart[1])  THEN
						
						(* Renan Added 10Jul26 - Puck Locker *)
						IF bPuckLockerEnable THEN
							GVL_Stations.stPuckLocker.nRequestedRelease 		:= USINT#1;
							GVL_Stations.stPuckLocker.bApplyDisposition 		:= TRUE;
						END_IF
						(*\Renan Added 10Jul26 - Puck Locker *)
						
						eCycleState												:= E_General_ProcessCycle.NEST_CLEARING;
						
					ELSIF ctuRejectPart.CV > 0 AND (bPartPresentNest1 OR (NOT bPartPresentNest2 AND bProcessedPart[1])) THEN
						
						bRejectPartFault										:= TRUE; 
					
					END_IF
					
					IF NOT bPartPresentNest2 AND bProcessedPart[1] THEN
						
						bRejectPartDialog[0]									:= TRUE;		
						sMachineMessage											:= 'WRONG PART TAKEN';
						
					ELSIF  bPartPresentNest2 THEN
						
						bRejectPartDialog[0]									:= FALSE;
						
					END_IF					
					
				ELSIF NOT stCycleDataNest1.bFail AND stCycleDataNest2.bFail THEN
					
					sMachineMessage												:= 'REMOVE PART FROM NEST 2 AND PUT IN REJECT CHUTE';
					
					IF ctuRejectPart.CV > 0 AND NOT bPartPresentNest2 AND (bPartPresentNest1 OR NOT bProcessedPart[0])  THEN
						
						(* Renan Added 10Jul26 - Puck Locker *)
						IF bPuckLockerEnable THEN
							GVL_Stations.stPuckLocker.nRequestedRelease 		:= USINT#1;
							GVL_Stations.stPuckLocker.bApplyDisposition 		:= TRUE;
						END_IF
						(*\Renan Added 10Jul26 - Puck Locker *)
						
						
						eCycleState												:= E_General_ProcessCycle.NEST_CLEARING;
						
					ELSIF ctuRejectPart.CV > 0 AND (bPartPresentNest1 OR (NOT bPartPresentNest1 AND bProcessedPart[0])) THEN
						
						bRejectPartFault										:= TRUE; 
					
					END_IF
					
					IF NOT bPartPresentNest1 AND bProcessedPart[0] THEN
						
						bRejectPartDialog[1]									:= TRUE;		
						sMachineMessage											:= 'WRONG PART TAKEN';
						
					ELSIF  bPartPresentNest1 THEN
						
						bRejectPartDialog[1]									:= FALSE;
						
					END_IF
				
				ELSIF stCycleDataNest1.bFail AND stCycleDataNest2.bFail THEN
					
					IF ctuRejectPart.CV > 1 AND NOT bPartPresentNest1 AND NOT bPartPresentNest2 THEN
						
						(* Renan Added 10Jul26 - Puck Locker *)
						IF bPuckLockerEnable THEN
							GVL_Stations.stPuckLocker.nRequestedRelease 		:= USINT#0;
							GVL_Stations.stPuckLocker.bApplyDisposition 		:= TRUE;
						END_IF
						(*\Renan Added 10Jul26 - Puck Locker *)
						
						eCycleState												:= E_General_ProcessCycle.NEST_CLEARING;
					
					ELSIF ctuRejectPart.CV > 1 AND ( bPartPresentNest1 OR bPartPresentNest2) THEN
						
						bRejectPartFault										:= TRUE; 		
					
					END_IF;
					
					sMachineMessage												:= 'REMOVE PART FROM BOTH NESTS AND PUT IN REJECT CHUTE';
					
				END_IF
				
E_General_ProcessCycle.NEST_CLEARING:
				
				IF bPuckLockerEnable AND GVL_Stations.stPuckLocker.eState = E_PuckLockerState.WaitingForNestsEmpty THEN
				
					IF (bPartPresentNest1 AND bNest1Flag) OR (bPartPresentNest2 AND bNest2Flag) THEN
						
						sMachineMessage 										:= 'Remove parts from nests to release puck';
						
					ELSE
						
						sMachineMessage 										:= 'Waiting for puck to be released';
						
					END_IF
				
				ELSIF (bPartPresentNest1 AND bNest1Flag) AND NOT (bPartPresentNest2 AND bNest2Flag)  THEN
					
					IF bPuckLockerEnable THEN
						
						sMachineMessage 										:= 'Remove processed part from nest 1 to release puck';
						
					ELSE
						
						sMachineMessage 										:= 'Remove Processed part from nest 1';
						
					END_IF
					
				ELSIF NOT (bPartPresentNest1 AND bNest1Flag) AND (bPartPresentNest2 AND bNest2Flag)  THEN 
					
					IF bPuckLockerEnable THEN
						
						sMachineMessage 										:= 'Remove processed part from nest 2 to release puck';
						
					ELSE
						
						sMachineMessage 										:= 'Remove Processed part from nest 2';
						
					END_IF
					
				ELSIF (bPartPresentNest1 AND bNest1Flag) AND (bPartPresentNest2 AND bNest2Flag) THEN 
					
					IF bPuckLockerEnable THEN
						
						sMachineMessage 										:= 'Remove processed parts to release puck';
						
					ELSE
						
						sMachineMessage 										:= 'Remove Processed parts';
						
					END_IF
					
				ELSIF (NOT bPartPresentNest1 OR NOT bNest1Flag) AND (NOT bPartPresentNest2 OR NOT bNest2Flag)  THEN
					
					sMachineMessage 											:= '';
					eCycleState													:= E_General_ProcessCycle.RESET_ALL_CMD;
									
				END_IF
				
END_CASE
END_ACTION

ACTION c_ACT_SaveData:

//SAVING NEST 1 DATA
IF bProcessedPart[0] THEN
	
	stCycleDataNest1.sDistance1				:= REAL_TO_STRING(stCycleDataNest1.HeightTest_anDistancesResult[1]);
	stCycleDataNest1.sDistance2				:= REAL_TO_STRING(stCycleDataNest1.HeightTest_anDistancesResult[2]);
	stCycleDataNest1.sDistance3				:= REAL_TO_STRING(stCycleDataNest1.HeightTest_anDistancesResult[3]);
	
	stCycleDataNest1.sSetpoint1				:= REAL_TO_STRING(stCycleDataNest1.HeightTest_anSetPoint[1]);
	stCycleDataNest1.sSetpoint2				:= REAL_TO_STRING(stCycleDataNest1.HeightTest_anSetPoint[2]);
	stCycleDataNest1.sSetpoint3				:= REAL_TO_STRING(stCycleDataNest1.HeightTest_anSetPoint[3]);
	
	IF stCycleDataNest1.bPass THEN
	
		stCycleDataNest1.sGeneralResult			:= 'PASS';

	ELSIF stCycleDataNest1.bFail THEN
	
		stCycleDataNest1.sGeneralResult			:= 'FAIL';

	END_IF

	IF stCycleDataNest1.HeightTest_Pass THEN
	
		stCycleDataNest1.sHeightTestResult		:= 'PASS';
	
	ELSIF stCycleDataNest1.HeightTest_Fail THEN
	
		stCycleDataNest1.sHeightTestResult		:= 'FAIL';
	
	END_IF



	IF stCycleDataNest1.LeakTest_Pass THEN
	
		stCycleDataNest1.sLeakTesterResult		:= 'PASS';

	ELSIF stCycleDataNest1.LeakTest_Fail THEN
	
		stCycleDataNest1.sLeakTesterResult		:= 'FAIL';
	
	END_IF
	
	aDataHistoryNest1[0]						:= stCycleDataNest1;
	
END_IF
	

//SAVING NEST 2 DATA

IF bProcessedPart[1] THEN
	
	stCycleDataNest2.sDistance1				:= REAL_TO_STRING(stCycleDataNest2.HeightTest_anDistancesResult[1]);
	stCycleDataNest2.sDistance2				:= REAL_TO_STRING(stCycleDataNest2.HeightTest_anDistancesResult[2]);
	stCycleDataNest2.sDistance3				:= REAL_TO_STRING(stCycleDataNest2.HeightTest_anDistancesResult[3]);
	
	stCycleDataNest2.sSetpoint1				:= REAL_TO_STRING(stCycleDataNest2.HeightTest_anSetPoint[1]);
	stCycleDataNest2.sSetpoint2				:= REAL_TO_STRING(stCycleDataNest2.HeightTest_anSetPoint[2]);
	stCycleDataNest2.sSetpoint3				:= REAL_TO_STRING(stCycleDataNest2.HeightTest_anSetPoint[3]);
	
	IF stCycleDataNest2.bPass THEN
	
		stCycleDataNest2.sGeneralResult			:= 'PASS';

	ELSIF stCycleDataNest2.bFail THEN
	
		stCycleDataNest2.sGeneralResult			:= 'FAIL';

	END_IF

	IF stCycleDataNest2.HeightTest_Pass THEN
	
		stCycleDataNest2.sHeightTestResult		:= 'PASS';
	
	ELSIF stCycleDataNest2.HeightTest_Fail THEN
	
		stCycleDataNest2.sHeightTestResult		:= 'FAIL';
	
	END_IF



	IF stCycleDataNest2.LeakTest_Pass THEN
	
		stCycleDataNest2.sLeakTesterResult		:= 'PASS';

	ELSIF stCycleDataNest2.LeakTest_Fail THEN
	
		stCycleDataNest2.sLeakTesterResult		:= 'FAIL';
	
	END_IF
	
	aDataHistoryNest2[0]						:= stCycleDataNest2;
	
END_IF
END_ACTION

ACTION d_ACT_IO:
//INPUTS

bPartPresentNest1					:= dw_T08_EL1809.iPartPresentNest1;
bPartPresentNest2					:= dw_T08_EL1809.iPartPresentNest2;

rRejectSensor( CLK := dw_T08_EL1809.iRejectSensor);

bDoorClosingFlag					:= (eCycleState = E_General_ProcessCycle.CLOSE_PROCESS_DOOR) OR (eCycleState = E_General_ProcessCycle.WAIT_CLOSE_PROCESS_DOOR) OR 
										bDoorClosingInitFlag;
bDoorOpeningFlag					:= eCycleState = E_General_ProcessCycle.OPEN_PROCESS_DOOR;

bProcessDoorClosedConditionFlag		:=  eCycleState = E_General_ProcessCycle.EXTEND_PROCESS_CYLINDER OR
										eCycleState = E_General_ProcessCycle.RETRACT_MIDDLE_PROCESS_CYLINDER OR
										eCycleState = E_General_ProcessCycle.WAIT_RETRACT_MIDDLE_PROCESS_CYLINDER OR
										eCycleState = E_General_ProcessCycle.LEAK_TEST OR
										eCycleState = E_General_ProcessCycle.WAIT_LEAK_TEST OR
										eCycleState = E_General_ProcessCycle.HEIGHT_TEST OR
										eCycleState = E_General_ProcessCycle.WAIT_HEIGHT_TEST OR
										eCycleState = E_General_ProcessCycle.RESULTS OR
										eCycleState = E_General_ProcessCycle.MOVE_NEST_TO_RIGHT OR
										eCycleState = E_General_ProcessCycle.WAIT_MOVE_NEST_TO_RIGHT OR
										eCycleState = E_General_ProcessCycle.MOVE_NEST_TO_LEFT OR
										eCycleState = E_General_ProcessCycle.WAIT_MOVE_NEST_TO_LEFT OR
										eCycleState = E_General_ProcessCycle.WAIT_TO_SAVE_DATA OR
										eCycleState = E_General_ProcessCycle.SAVE_DATA OR
										eCycleState = E_General_ProcessCycle.SAVE_DATA2 OR
										eCycleState = E_General_ProcessCycle.CSV_NEST1 OR
										eCycleState = E_General_ProcessCycle.CSV_NEST2 OR
										eCycleState = E_General_ProcessCycle.RETRACT_PROCESS_CYLINDER OR
										eCycleState = E_General_ProcessCycle.WAIT_RETRACT_PROCESS_CYLINDER;
					

										

										
tonTwoHandsSignal( IN := stTwinSAFE.qTwoHandsSafe , PT := stTimers.tTwoHandsSignal);						
				
bTwoHandsSignal						:= tonTwoHandsSignal.Q;
		
dw_T09_EL2809.qIndicatorLED1_Red	:= stCycleDataNest1.bFail;		
dw_T09_EL2809.qIndicatorLED1_Green	:= stCycleDataNest1.bPass;	
dw_T09_EL2809.qIndicatorLED2_Red	:= stCycleDataNest2.bFail;		
dw_T09_EL2809.qIndicatorLED2_Green	:= stCycleDataNest2.bPass;	

IF 	(stMachineStatus.eMachineState = E_MachineState.SYSTEM_AUTO_CYCLE) AND NOT ((eCycleState	= E_General_ProcessCycle.IDLE) OR eCycleState	= E_General_ProcessCycle.WAIT_REJECT_PART) THEN
	

	bPartPresent[0]					:= 	bProcessedPart[0];
	bPartPresent[1]					:= 	bProcessedPart[1];
	
ELSE	
		bPartPresent[0]				:= dw_T08_EL1809.iPartPresentNest1;
		bPartPresent[1]				:= dw_T08_EL1809.iPartPresentNest2;

END_IF
				
stTwinSAFE.iMachineHoming_Manual		:= 	stMachineStatus.eMachineState = E_MachineState.SAFETY OR
										stMachineStatus.eMachineState = E_MachineState.SYSTEM_INITIALISING OR 
										stMachineStatus.eMachineState = E_MachineState.MANUAL_MODE;												
										
bSlideNestNotHomed					:= NOT dw_T08_EL1809.iSlideNestRetracted;

dw_T09_EL2809.qTopSealer			:= bTopSealer OR (stMachineStatus.bManualMode AND bTopSealer_HMI);												
dw_T09_EL2809.qBottomSealer			:= bBottomSealer OR (stMachineStatus.bManualMode AND bBottomSealer_HMI);
END_ACTION

END_PROGRAM
